PROGRAM UnitTests
VAR
    pidTests : Pid_Tests;
END_VAR

TcUnit.RUN();

END_PROGRAM

(* stored: Version 1.1.0.1, ProductVersion 3.1.4024.11
   POU UnitTests: Id {dde40bb1-b2ba-43e6-8c92-b0dedcf8ee20}, SpecialFunc None *)
